FUNCTION_BLOCK FB_Conveyor EXTENDS FB_Generic
VAR
	bExecuteComplete: BOOL;
	nStateChanges	: INT;
END_VAR

SUPER^();

{attribute 'object_name' := 'M_Execute'}
METHOD M_Execute
IF bExecuteComplete THEN
	bExecuteComplete := FALSE;
	M_StateComplete();
END_IF
END_METHOD

{attribute 'object_name' := 'M_Resetting'}
METHOD M_Resetting
VAR_INST
	delay	: TON;
END_VAR
delay( IN := NOT delay.Q, PT := T#2S );

IF delay.Q THEN
	THIS^.M_StateComplete();
END_IF
END_METHOD

{attribute 'object_name' := 'M_StateComplete'}
METHOD M_StateComplete
nStateChanges := nStateChanges + 1;
SUPER^.M_StateComplete();
END_METHOD

END_FUNCTION_BLOCK

(* stored: Version 1.1.0.1, ProductVersion 3.1.4024.10
   POU FB_Conveyor: Id {9df1c638-35b3-49a7-b21b-402a6466bb05}, SpecialFunc None
   Method M_Execute: Id {8742ee40-11c8-4a3a-8440-d53d83ebace3}
   Method M_Resetting: Id {ab1acdfd-3a9a-4b1d-b99f-106863350fe2}
   Method M_StateComplete: Id {95201eb5-7bf4-4247-b3f1-01ab3a380f58} *)
